VAR_GLOBAL


END_VAR

(* stored: Version 1.1.0.1, ProductVersion 3.1.4022.18
   GVL GVL_MOT: Id {0bf73307-23cf-49fa-b7ca-fc54da613ef3} *)
